         // Nach der Anwahl des Referenziertyps "Fliegendes Referenzieren", 
         // ein Zyklus später kann das Referenzieren gestartet
         IF (#siRefTypCyc = 0) THEN
           #siRefTypCyc := #siRefTypCyc + 1;
         ELSE
           // Referenzieren starten
           //#sxSendBuf.sxSTW1.RefStart := True;
           #sxSendBuf.STW1.%X11 := True;
         END_IF;
       END_IF;
     END_IF;
   ELSE
     // Werte wieder zurücknehmen
     (*#sxSendBuf.sxSTW1.Off1          := #Off1;
             #sxSendBuf.sxSTW1.RejTrvTsk     := False;
             #sxSendBuf.sxSTW1.TrvStart      := False;
             #sxSendBuf.sxEPosSTW1.MdiStart  := False;
             #sxSendBuf.sxSTW1.Jog1          := False;
             #sxSendBuf.sxSTW1.Jog2          := False;
             #sxSendBuf.sxEPosSTW1.MdiTyp    := False;
             #sxSendBuf.sxEPosSTW1.MdiPos    := False;
             #sxSendBuf.sxEPosSTW1.MdiNeg    := False;
             #sxSendBuf.sxEPosSTW1.MdiTrTyp  := False;
             #sxSendBuf.sxEPosSTW1.MdiSetup  := False;
             #sxSendBuf.sxEPosSTW2.SetRefPt  := False;
             #sxSendBuf.sxEPosSTW2.RefTyp    := False;
             #sxSendBuf.sxEPosSTW2.RefStDi   := False;
             #sxSendBuf.sxEPosSTW2.JogInc    := False;
             #sxSendBuf.sxSTW1.RefStart      := False;*)

     #sxSendBuf.STW1.%X0 := #EnableAxis;
     #sxSendBuf.STW1.%X4 := False;
     #sxSendBuf.STW1.%X6 := False;
     #sxSendBuf.EPosSTW1.%X15 := False;
     #sxSendBuf.STW1.%X8 := False;
     #sxSendBuf.STW1.%X9 := False;
     #sxSendBuf.EPosSTW1.%X8 := False;
     #sxSendBuf.EPosSTW1.%X9 := False;
     #sxSendBuf.EPosSTW1.%X10 := False;
     #sxSendBuf.EPosSTW1.%X12 := False;
     #sxSendBuf.EPosSTW1.%X14 := False;
     #sxSendBuf.EPosSTW2.%X1 := False;
     #sxSendBuf.EPosSTW2.%X8 := False;
     #sxSendBuf.EPosSTW2.%X9 := False;
     #sxSendBuf.EPosSTW2.%X5 := False;
     #sxSendBuf.STW1.%X11 := False;
   END_IF; // Hauptbetriebsart "Verfahrsätze" (Traversing Blocks)

   //Den Eingang ConfigEPos auf die einzelnen Bits im Telegramm verschalten
   #sxSendBuf.STW1.%X1 := #ConfigEPos.%X0;
   #sxSendBuf.STW1.%X2 := #ConfigEPos.%X1;
   #sxSendBuf.EPosSTW2.%X14 := #ConfigEPos.%X2;
   #sxSendBuf.EPosSTW2.%X15 := #ConfigEPos.%X3;
   #sxSendBuf.EPosSTW2.%X11 := #ConfigEPos.%X4;
   #sxSendBuf.EPosSTW2.%X10 := #ConfigEPos.%X5;
   #sxSendBuf.EPosSTW2.%X2 := #ConfigEPos.%X6;
   #sxSendBuf.STW1.%X13 := #ConfigEPos.%X7;
   #sxSendBuf.EPosSTW1.%X12 := #ConfigEPos.%X8;
   #sxSendBuf.STW2.%X0 := #ConfigEPos.%X9;
   #sxSendBuf.STW2.%X1 := #ConfigEPos.%X10;
   #sxSendBuf.STW2.%X2 := #ConfigEPos.%X11;
   #sxSendBuf.STW2.%X3 := #ConfigEPos.%X12;
   #sxSendBuf.STW2.%X4 := #ConfigEPos.%X13;
   #sxSendBuf.STW2.%X7 := #ConfigEPos.%X14;
   #sxSendBuf.STW1.%X12 := #ConfigEPos.%X15;
   #sxSendBuf.STW1.%X14 := #ConfigEPos.%X16;
   #sxSendBuf.STW1.%X15 := #ConfigEPos.%X17;
   #sxSendBuf.EPosSTW1.%X6 := #ConfigEPos.%X18;
   #sxSendBuf.EPosSTW1.%X7 := #ConfigEPos.%X19;
   #sxSendBuf.EPosSTW1.%X11 := #ConfigEPos.%X20;
   #sxSendBuf.EPosSTW1.%X13 := #ConfigEPos.%X21;
   #sxSendBuf.EPosSTW2.%X3 := #ConfigEPos.%X22;
   #sxSendBuf.EPosSTW2.%X4 := #ConfigEPos.%X23;
   #sxSendBuf.EPosSTW2.%X6 := #ConfigEPos.%X24;
   #sxSendBuf.EPosSTW2.%X7 := #ConfigEPos.%X25;
   #sxSendBuf.EPosSTW2.%X12 := #ConfigEPos.%X26;
   #sxSendBuf.EPosSTW2.%X13 := #ConfigEPos.%X27;
   #sxSendBuf.STW2.%X5 := #ConfigEPos.%X28;
   #sxSendBuf.STW2.%X6 := #ConfigEPos.%X29;
   #sxSendBuf.STW2.%X8 := #ConfigEPos.%X30;
   #sxSendBuf.STW2.%X9 := #ConfigEPos.%X31;


   #swSendBuf[0] := #sxSendBuf.STW1;
   #swSendBuf[1] := #sxSendBuf.EPosSTW1;
   #swSendBuf[2] := #sxSendBuf.EPosSTW2;
   #swSendBuf[3] := #sxSendBuf.STW2;
   #swSendBuf[4] := #sxSendBuf.OverrideV;
   #swSendBuf[5] := #sxSendBuf.Position.%W1;
   #swSendBuf[6] := #sxSendBuf.Position.%W0;
   #swSendBuf[7] := #sxSendBuf.Velocity.%W1;
   #swSendBuf[8] := #sxSendBuf.Velocity.%W0;
   #swSendBuf[9] := #sxSendBuf.OverrideA;
   #swSendBuf[10] := #sxSendBuf.OverrideD;
   #swSendBuf[11] := #sxSendBuf.Reserve;

   //Prozessdaten zur Signalbaugruppe schreiben
   #piRetSFC := DPWR_DAT(LADDR := #HWIDSTW,
                         RECORD := #swSendBuf);

   // Fehler der Rückmeldung ausgeben
   #DiagID := INT_TO_WORD(#piRetSFC);

   //kein Fehler beim Schreiben
   IF #piRetSFC = 0 THEN

     // Fehler wieder zurück nehmen
     IF (#swStatus = 16#8601) THEN
       #swStatus := 16#7002;
       #Error := False;
     END_IF;

     //Prozessdaten von der Signalbaugruppe lesen
     #piRetSFC := DPRD_DAT(LADDR := #HWIDZSW,
                           RECORD => #swRecvBuf);

     // Fehlermeldung der Rückmeldung ausgeben
     #DiagID := INT_TO_WORD(#piRetSFC);

     //Fehler beim Lesen (Profibus-Kommunikation unterbrochen)
     IF #piRetSFC <> 0 THEN

       // Fehler
       #Error := TRUE;
       #swStatus := 16#8600;

       // Zustandsworte löschen
       #sxRecvBuf.ZSW1 := W#16#0;
       #sxRecvBuf.EPosZSW1 := W#16#0;
       #sxRecvBuf.EPosZSW2 := W#16#0;
       #sxRecvBuf.ZSW2 := W#16#0;
       #sxRecvBuf.NotUsed := W#16#00;
       #sxRecvBuf.Position := DW#16#00;
       #sxRecvBuf.Velocity := DW#16#00;
       #sxRecvBuf.ErrNr := W#16#00;
       #sxRecvBuf.WarnNr := W#16#00;
       #sxRecvBuf.Reserve := W#16#00;

       // Werte auslesen
     ELSE

       // Fehler wieder zurück nehmen
       IF (#swStatus = 16#8600) THEN
         #swStatus := 16#7002;
         #Error := False;
       END_IF;

       #sxRecvBuf.ZSW1 := #swRecvBuf[0];
       #sxRecvBuf.EPosZSW1 := #swRecvBuf[1];
       #sxRecvBuf.EPosZSW2 := #swRecvBuf[2];
       #sxRecvBuf.ZSW2 := #swRecvBuf[3];
       #sxRecvBuf.NotUsed := #swRecvBuf[4];
       #sxRecvBuf.Position.%W1 := #swRecvBuf[5];
       #sxRecvBuf.Position.%W0 := #swRecvBuf[6];
       #sxRecvBuf.Velocity.%W1 := #swRecvBuf[7];
       #sxRecvBuf.Velocity.%W0 := #swRecvBuf[8];
       #sxRecvBuf.ErrNr := #swRecvBuf[9];
       #sxRecvBuf.WarnNr := #swRecvBuf[10];
       #sxRecvBuf.Reserve := #swRecvBuf[11];

       #aaa := INT_TO_REAL(WORD_TO_INT(#sxRecvBuf.Reserve));
       #bbb:=NORM_X_REAL(MAX := 16384.0, MIN := -16384.0, VALUE := #aaa);
       #Torque :=ABS(SCALE_X_REAL(MIN := #RefTorque*-1, MAX :=#RefTorque, VALUE := #bbb));

       // ZSW1 aufbereiten
       //#Busy := #sxRecvBuf.sxZSW1.IOp;
       #sbBusy := #sxRecvBuf.ZSW1.%X2;

       // Fehler auswerten
       IF #sxRecvBuf.ZSW1.%X3 THEN
           #swStatus := 16#8401;
         #Error := True;
       ELSIF #sxRecvBuf.ZSW1.%X6 THEN
         #swStatus := 16#8402;
         #Error := True;
       ELSE
         // Fehler wieder zurück nehmen
         IF (#swStatus = 16#8401) OR (#swStatus = 16#8402) THEN
           #swStatus := 16#7002;
           #Error := False;
         END_IF;
       END_IF;

       // EPOS_ZSW1            
       // EPOS-Wort-1 BIT 00 --> 1 = Active traversing block bit 0
       //IF #sxRecvBuf.sxEPosZSW1.ActTrvBit0 THEN
       IF #sxRecvBuf.EPosZSW1.%X0 THEN
         #swEPosZSW1 := #swEPosZSW1 OR W#16#01;
       ELSE
         #swEPosZSW1 := #swEPosZSW1 AND W#16#FFFE;
       END_IF;

       // EPOS-Wort-1 Bit 01 --> 1 = Active traversing block bit 1
       //IF #sxRecvBuf.sxEPosZSW1.ActTrvBit1 THEN
       IF #sxRecvBuf.EPosZSW1.%X1 THEN
         #swEPosZSW1 := #swEPosZSW1 OR W#16#02;
       ELSE
         #swEPosZSW1 := #swEPosZSW1 AND W#16#FFFD;
       END_IF;

       // EPOS-Wort-1 Bit 02 --> 1 = Active traversing block bit 2
       //IF #sxRecvBuf.sxEPosZSW1.ActTrvBit2 THEN
       IF #sxRecvBuf.EPosZSW1.%X2 THEN
         #swEPosZSW1 := #swEPosZSW1 OR W#16#04;
       ELSE
         #swEPosZSW1 := #swEPosZSW1 AND W#16#FFFB;
       END_IF;

       // EPOS-Wort-1 Bit 03 --> 1 = Active traversing block bit 3
       //IF #sxRecvBuf.sxEPosZSW1.ActTrvBit3 THEN
       IF #sxRecvBuf.EPosZSW1.%X3 THEN
         #swEPosZSW1 := #swEPosZSW1 OR W#16#08;
       ELSE
         #swEPosZSW1 := #swEPosZSW1 AND W#16#FFF7;
       END_IF;

       // EPOS-Wort-1 Bit 04 --> 1 = Active traversing block bit 4 
       //IF #sxRecvBuf.sxEPosZSW1.ActTrvBit4 THEN
       IF #sxRecvBuf.EPosZSW1.%X4 THEN
         #swEPosZSW1 := #swEPosZSW1 OR W#16#10;
       ELSE
         #swEPosZSW1 := #swEPosZSW1 AND W#16#FFEF;
       END_IF;

       // EPOS-Wort-1 Bit 05 --> 1 = Active traversing block bit 5
       //IF #sxRecvBuf.sxEPosZSW1.ActTrvBit5 THEN
       IF #sxRecvBuf.EPosZSW1.%X5 THEN
         #swEPosZSW1 := #swEPosZSW1 OR W#16#20;
       ELSE
         #swEPosZSW1 := #swEPosZSW1 AND W#16#FFDF;
       END_IF;

       // EPOS-Wort-1 Bit 08 --> 1 = STOP cam minus active
       //IF #sxRecvBuf.sxEPosZSW1.StpCamMinAct THEN
       IF #sxRecvBuf.EPosZSW1.%X8 THEN
         #swEPosZSW1 := #swEPosZSW1 OR W#16#100;
       ELSE
         #swEPosZSW1 := #swEPosZSW1 AND W#16#FEFF;
       END_IF;

       // EPOS-Wort-1 Bit 09 --> 1 = STOP cam plus active
       //IF #sxRecvBuf.sxEPosZSW1.StpCamPlsAct THEN
       IF #sxRecvBuf.EPosZSW1.%X9 THEN
         #swEPosZSW1 := #swEPosZSW1 OR W#16#200;
       ELSE
         #swEPosZSW1 := #swEPosZSW1 AND W#16#FDFF;
       END_IF;

       // EPOS-Wort-1 Bit 10 --> 1 = Jogging active
       //IF #sxRecvBuf.sxEPosZSW1.JogAct THEN
       IF #sxRecvBuf.EPosZSW1.%X10 THEN
         #swEPosZSW1 := #swEPosZSW1 OR W#16#400;
       ELSE
         #swEPosZSW1 := #swEPosZSW1 AND W#16#FBFF;
       END_IF;

       // EPOS-Wort-1 Bit 11 --> 1 = Reference point approach active
       //IF #sxRecvBuf.sxEPosZSW1.RefAct THEN
       IF #sxRecvBuf.EPosZSW1.%X11 THEN
         #swEPosZSW1 := #swEPosZSW1 OR W#16#800;
       ELSE
         #swEPosZSW1 := #swEPosZSW1 AND W#16#F7FF;
       END_IF;

       // Anstossen des fliegenden Referenzieren prüfen, wenn die Rückmeldung fehlt dann wiederholen
       //IF NOT #sxRecvBuf.sxEPosZSW1.FlyRefAct AND #sbRefTyp AND #sxSendBuf.sxSTW1.RefStart THEN
       IF NOT #sxRecvBuf.EPosZSW1.%X12 AND #sbRefTyp AND #sxSendBuf.STW1.%X11 THEN

         // Wiederholung anstossen 
         IF #siRefActRetry < #siRetryMax THEN
           #siRefActRetry := #siRefActRetry + 1;

           // Referenzieren starten wieder wegnehmen
           //#sxSendBuf.sxSTW1.RefStart := False;
           #sxSendBuf.STW1.%X11 := False;
         ELSE

           // Fehlermeldung
           #swStatus := 16#8403;
           #Error := True;
         END_IF;
       ELSE

         // Fehler wieder zurücknehmen, wenn er mal ausgelöst wurde
         IF #swStatus = 16#8403 THEN
           #swStatus := 16#7002;
           #Error := False;
         END_IF;
         // Zähler zurücksetzen bei Rückmeldung fliegendes Referenzieren jetzt aktiviert oder bei Abwahl der Funktion
         IF (#sxRecvBuf.EPosZSW1.%X12 AND #sbRefTyp AND #sxSendBuf.STW1.%X11) OR NOT #FlyRef THEN
           #siRefActRetry := 0;
         END_IF;
       END_IF;

       // EPOS-Wort-1 Bit 12 --> 1 = Flying referencing active
       //IF #sxRecvBuf.sxEPosZSW1.FlyRefAct THEN
       IF #sxRecvBuf.EPosZSW1.%X12 THEN
         #swEPosZSW1 := #swEPosZSW1 OR W#16#1000;
       ELSE
         #swEPosZSW1 := #swEPosZSW1 AND W#16#EFFF;
       END_IF;

       // EPOS-Wort-1 Bit 13 --> 1 = Traversing block active
       //IF #sxRecvBuf.sxEPosZSW1.TrvBlAct THEN
       IF #sxRecvBuf.EPosZSW1.%X13 THEN
         #swEPosZSW1 := #swEPosZSW1 OR W#16#2000;
       ELSE
         #swEPosZSW1 := #swEPosZSW1 AND W#16#DFFF;
       END_IF;

       // EPOS-Wort-1 Bit 14 --> 1 = MDI setup active
       //IF #sxRecvBuf.sxEPosZSW1.MdiStupAct THEN
       IF #sxRecvBuf.EPosZSW1.%X14 THEN
         #swEPosZSW1 := #swEPosZSW1 OR W#16#4000;
       ELSE
         #swEPosZSW1 := #swEPosZSW1 AND W#16#BFFF;
       END_IF;

       // EPOS-Wort-1 Bit 15 --> 1 = MDI positing active
       //IF #sxRecvBuf.sxEPosZSW1.MdiPosAct THEN
       IF #sxRecvBuf.EPosZSW1.%X15 THEN
         #swEPosZSW1 := #swEPosZSW1 OR W#16#8000;
       ELSE
         #swEPosZSW1 := #swEPosZSW1 AND W#16#7FFF;
       END_IF;

       // EPOS_ZSW2 
       // EPOS-Wort-2 Bit 00 --> 1 = Tracking mode active
       //IF #sxRecvBuf.sxEPosZSW2.TrkModeAct THEN
       IF #sxRecvBuf.EPosZSW2.%X0 THEN
         #swEPosZSW2 := #swEPosZSW2 OR W#16#01;
       ELSE
         #swEPosZSW2 := #swEPosZSW2 AND W#16#FFFE;
       END_IF;

       // EPOS-Wort-2 Bit 01 --> 1 = Velocity limit active
       //IF #sxRecvBuf.sxEPosZSW2.VeloLimAct THEN
       IF #sxRecvBuf.EPosZSW2.%X1 THEN
         #swEPosZSW2 := #swEPosZSW2 OR W#16#02;
       ELSE
         #swEPosZSW2 := #swEPosZSW2 AND W#16#FFFD;
       END_IF;

       // EPOS-Wort-2 Bit 02 --> 1 = Setpoint static
       //IF #sxRecvBuf.sxEPosZSW2.SetPStat THEN
       IF #sxRecvBuf.EPosZSW2.%X2 THEN
         #swEPosZSW2 := #swEPosZSW2 OR W#16#04;
       ELSE
         #swEPosZSW2 := #swEPosZSW2 AND W#16#FFFB;
       END_IF;

       // EPOS-Wort-2 Bit 03 --> 1 = Printmark outside outer window
       //IF #sxRecvBuf.sxEPosZSW2.PrnMrkOut THEN
       IF #sxRecvBuf.EPosZSW2.%X3 THEN
         #swEPosZSW2 := #swEPosZSW2 OR W#16#08;
       ELSE
         #swEPosZSW2 := #swEPosZSW2 AND W#16#FFF7;
       END_IF;

       // EPOS-Wort-2 Bit 04 --> 1 = Axis forwards
       //IF #sxRecvBuf.sxEPosZSW2.FWD THEN
       IF #sxRecvBuf.EPosZSW2.%X4 THEN
         #swEPosZSW2 := #swEPosZSW2 OR W#16#10;
       ELSE
         #swEPosZSW2 := #swEPosZSW2 AND W#16#FFEF;
       END_IF;

       // EPOS-Wort-2 Bit 05 --> 1 = Axis backwards
       //IF #sxRecvBuf.sxEPosZSW2.BWD THEN
       IF #sxRecvBuf.EPosZSW2.%X5 THEN
         #swEPosZSW2 := #swEPosZSW2 OR W#16#20;
       ELSE
         #swEPosZSW2 := #swEPosZSW2 AND W#16#FFDF;
       END_IF;

       // EPOS-Wort-2 Bit 06 --> 1 = Software limit switch minus active
       //IF #sxRecvBuf.sxEPosZSW2.SftSwMinAct THEN
       IF #sxRecvBuf.EPosZSW2.%X6 THEN
         #swEPosZSW2 := #swEPosZSW2 OR W#16#40;
       ELSE
         #swEPosZSW2 := #swEPosZSW2 AND W#16#FFBF;
       END_IF;

       // EPOS-Wort-2 Bit 07 --> 1 = Software limit switch plus active
       //IF #sxRecvBuf.sxEPosZSW2.SftSwPlsAct THEN
       IF #sxRecvBuf.EPosZSW2.%X7 THEN
         #swEPosZSW2 := #swEPosZSW2 OR W#16#80;
       ELSE
         #swEPosZSW2 := #swEPosZSW2 AND W#16#FF7F;
       END_IF;

       // EPOS-Wort-2 Bit 08 --> 1 = Position actual value <= cam position 1
       //IF #sxRecvBuf.sxEPosZSW2.PosSmCam1 THEN
       IF #sxRecvBuf.EPosZSW2.%X8 THEN
         #swEPosZSW2 := #swEPosZSW2 OR W#16#100;
       ELSE
         #swEPosZSW2 := #swEPosZSW2 AND W#16#FEFF;
       END_IF;

       // EPOS-Wort-2 Bit 09 --> 1 = Position actual value <= cam position 2
       //IF #sxRecvBuf.sxEPosZSW2.PosSmCam2 THEN
       IF #sxRecvBuf.EPosZSW2.%X9 THEN
         #swEPosZSW2 := #swEPosZSW2 OR W#16#200;
       ELSE
         #swEPosZSW2 := #swEPosZSW2 AND W#16#FDFF;
       END_IF;

       // EPOS-Wort-2 Bit 10 --> 1 = Direct output 1 via traversing block
       //IF #sxRecvBuf.sxEPosZSW2.TrvOut1 THEN
       IF #sxRecvBuf.EPosZSW2.%X10 THEN
         #swEPosZSW2 := #swEPosZSW2 OR W#16#400;
       ELSE
         #swEPosZSW2 := #swEPosZSW2 AND W#16#FBFF;
       END_IF;

       // EPOS-Wort-2 Bit 11 --> 1 = Direct output 2 via traversing block
       //IF #sxRecvBuf.sxEPosZSW2.TrvOut2 THEN
       IF #sxRecvBuf.EPosZSW2.%X11 THEN
         #swEPosZSW2 := #swEPosZSW2 OR W#16#800;
       ELSE
         #swEPosZSW2 := #swEPosZSW2 AND W#16#F7FF;
       END_IF;

       // EPOS-Wort-2 Bit 12 --> 1 = Fixed STOP reached
       //IF #sxRecvBuf.sxEPosZSW2.FxStpRd THEN
       IF #sxRecvBuf.EPosZSW2.%X12 THEN
         #swEPosZSW2 := #swEPosZSW2 OR W#16#1000;
       ELSE
         #swEPosZSW2 := #swEPosZSW2 AND W#16#EFFF;
       END_IF;

       // EPOS-Wort-2 Bit 13 --> 1 = Fixed STOP clamping torque reached
       //IF #sxRecvBuf.sxEPosZSW2.FxStpTrRd THEN
       IF #sxRecvBuf.EPosZSW2.%X13 THEN
         #swEPosZSW2 := #swEPosZSW2 OR W#16#2000;
       ELSE
         #swEPosZSW2 := #swEPosZSW2 AND W#16#DFFF;
       END_IF;

       // EPOS-Wort-2 Bit 14 --> 1 = Traversing fixed STOP active
       //IF #sxRecvBuf.sxEPosZSW2.TrvFxStpAct THEN
       IF #sxRecvBuf.EPosZSW2.%X14 THEN
         #swEPosZSW2 := #swEPosZSW2 OR W#16#4000;
       ELSE
         #swEPosZSW2 := #swEPosZSW2 AND W#16#BFFF;
       END_IF;

       // EPOS-Wort-2 Bit 15 --> 1 = Traversing command active
       //IF #sxRecvBuf.sxEPosZSW2.CmdAct THEN
       IF #sxRecvBuf.EPosZSW2.%X15 THEN
         #swEPosZSW2 := #swEPosZSW2 OR W#16#8000;
       ELSE
         #swEPosZSW2 := #swEPosZSW2 AND W#16#7FFF;
       END_IF;

       #sbReady := #sxRecvBuf.ZSW1.%X1;

       #AxisEnabled := #sxRecvBuf.ZSW1.%X2;
       #sbIOp := #sxRecvBuf.ZSW1.%X2;

       #AxisError := #sxRecvBuf.ZSW1.%X3;
       #sbFault := #sxRecvBuf.ZSW1.%X3;

       #AxisWarn := #sxRecvBuf.ZSW1.%X7;
       #sbAlarm := #sxRecvBuf.ZSW1.%X7;

       #AxisPosOk := #sxRecvBuf.ZSW1.%X10;
       #AxisRef := #sxRecvBuf.ZSW1.%X11;
       #AxisSpFixed := #sxRecvBuf.ZSW1.%X13;

       #sbAccel := #sxRecvBuf.ZSW1.%X14;
       #sbDecel := #sxRecvBuf.ZSW1.%X15;

       //#ActVelocity := DWORD_TO_DINT(#sxRecvBuf.Velocity);
       #v1 := DINT_TO_REAL(DWORD_TO_DINT(#sxRecvBuf.Velocity));
       #v2:=(#v1+16#40000000) / 16#80000000;
       #ActVelocity := ABS(SCALE_X_REAL(MIN := -1*#RefSpeed, MAX := #RefSpeed, VALUE := #v2));

       //#ActPosition := DWORD_TO_DINT(#sxRecvBuf.Position);
       #ActPosition :=(DINT_TO_REAL(DWORD_TO_DINT(#sxRecvBuf.Position)) / #Factor);


       #ActMode := #ModePos;
       #ActWarn := #sxRecvBuf.WarnNr;
       #ActFault := #sxRecvBuf.ErrNr;

       #Lockout := #sxRecvBuf.ZSW1.%X6;
       //Soft Positio OK
       IF ABS_REAL(#Position - #ActPosition) < #SoftPosTlr THEN
           ;
           #SoftPosOK := TRUE;
       ELSE
           #SoftPosOK := FALSE;
       END_IF;
     END_IF;
   ELSE

     // Fehler
     #Error := TRUE;
     #swStatus := 16#8601;

   END_IF;

   // Initialisierung von Ausg㭧en
   #Status := #swStatus;
   #EPosZSW1 := #swEPosZSW1;
   #EPosZSW2 := #swEPosZSW2;
END_FUNCTION_BLOCK

// ===== library: MasterCopy "ServoAxisV90" =====

// folder: AxisControl

FUNCTION_BLOCK "ServoAxisV90"   // FB602, LAD
{ S7_Optimized_Access := 'TRUE' }
VERSION : 0.1
   VAR_INPUT
      HwID : HW_IO;
      "Enb?" : Bool;
      iLLim : Bool;
      iHLim : Bool;
      iMotionPermit : Bool;
      iJogPermit : Bool;
      iReset : Bool;
      bwPos : Real := 0.0;   // Geri Pozisyon Bilgisi
      fwPos : Real := 0.0;   // İleri Pozisyon Bilgisi
      bwTol : Real := 0.0;   // İleride Bilgisi Toleransı
      fwTol : Real := 0.0;   // Geride Bilgisi Toleransı
      inSpeed : Real;
   END_VAR
   VAR_OUTPUT
      qBrake : Bool;
   END_VAR
   VAR_IN_OUT
      ManCmd : "ManServo";
      iHoldingOff : Bool;
   END_VAR
   VAR
      Servo : "SINA_POS";
      AutoCmd : Struct
         Go1TargetPos : Bool;
         Go2TargetPos : Bool;
         Go3TargetPos : Bool;
         Go1WaitingPos : Bool;
         Go2WaitingPos : Bool;
         Go3WaitingPos : Bool;
         Go4WaitingPos : Bool;
         TargetPos : Real;
         WaitingPos : Real;
         Speed : Int;
      END_STRUCT;
      Auto : Struct
         GoAbs : Bool;
         "Step" : Int;
      END_STRUCT;
      Man : Struct
         GoAbs : Bool;
         "Step" : Int;
      END_STRUCT;
      Homing : Struct
         Execute : Bool;
         "Step" : Int;
      END_STRUCT;
      Ready : Bool;
      OnSafetyArea : Bool;
      PosOK : Bool;
      OnBwPos : Bool;
      OnFwPos : Bool;
      OnBw2Pos : Bool;
      mAxisMoving : Bool;
      PosTemp : Real;
      "Timer" : Struct
         T1 : IEC_TIMER;
         T2 : IEC_TIMER;
         T3 : IEC_TIMER;
         T4 : IEC_TIMER;
         T5 : IEC_TIMER;
         T6 : IEC_TIMER;
         T7 : IEC_TIMER;
         T8 : IEC_TIMER;
         T9 : IEC_TIMER;
         T10 : IEC_TIMER;
         T11 : IEC_TIMER;
      END_STRUCT;
      Alarm : Struct
         PermissionErr : Bool;
         EnbErr : Bool;
      END_STRUCT;
      negBwTol : Real;
      p_trg : Array[0..3] of Bool;
      negFwTol : Real;
      ovDec : Int;
   END_VAR
   VAR_TEMP
      Temp1 : Real;
      Temp2 : Real;
      temp3 : Real;
   END_VAR
   VAR_TEMP   // added for the SCL form of the ladder/FBD networks
      _w1 : Bool;
      _w2 : Bool;
      _w3 : Bool;
      _w4 : Bool;
   END_VAR
BEGIN

REGION Network 1: Sina Pos Block
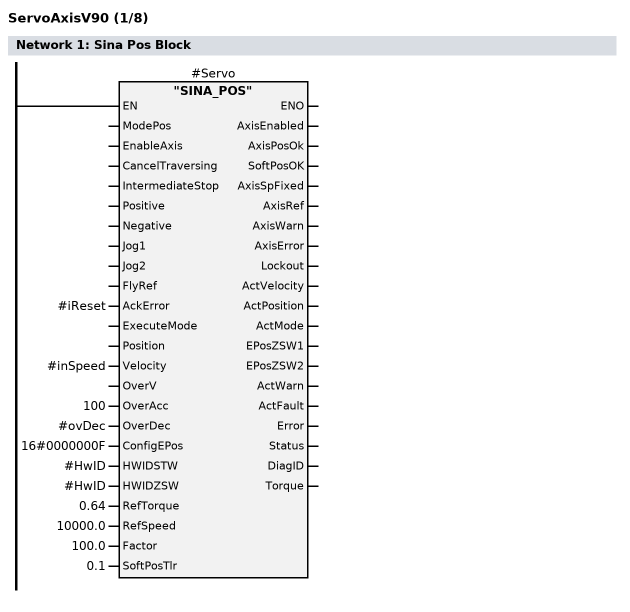
   RUNG wire#powerrail
      #Servo(ModePos :=, EnableAxis :=, CancelTraversing :=, IntermediateStop :=, Positive :=, Negative :=, Jog1 :=, Jog2 :=, FlyRef :=, AckError := #iReset, ExecuteMode :=, Position :=, Velocity := #inSpeed, OverV :=, OverAcc := 100, OverDec := #ovDec, ConfigEPos := 16#0000000F, HWIDSTW := #HwID, HWIDZSW := #HwID, RefTorque := 0.64, RefSpeed := 10000.0, Factor := 100.0, SoftPosTlr := 0.1, AxisEnabled =>, AxisPosOk =>, SoftPosOK =>, AxisSpFixed =>, AxisRef =>, AxisWarn =>, AxisError =>, Lockout =>, ActVelocity =>, ActPosition =>, ActMode =>, EPosZSW1 =>, EPosZSW2 =>, ActWarn =>, ActFault =>, Error =>, Status =>, DiagID =>, Torque =>)
   END_RUNG
   // the same network as SCL:
   #Servo(AckError := #iReset,   // "SINA_POS"
          Velocity := #inSpeed,
          OverAcc := 100,
          OverDec := #ovDec,
          ConfigEPos := 16#0000000F,
          HWIDSTW := #HwID,
          HWIDZSW := #HwID,
          RefTorque := 0.64,
          RefSpeed := 10000.0,
          Factor := 100.0,
          SoftPosTlr := 0.1);
END_REGION

REGION Network 2: Drive On
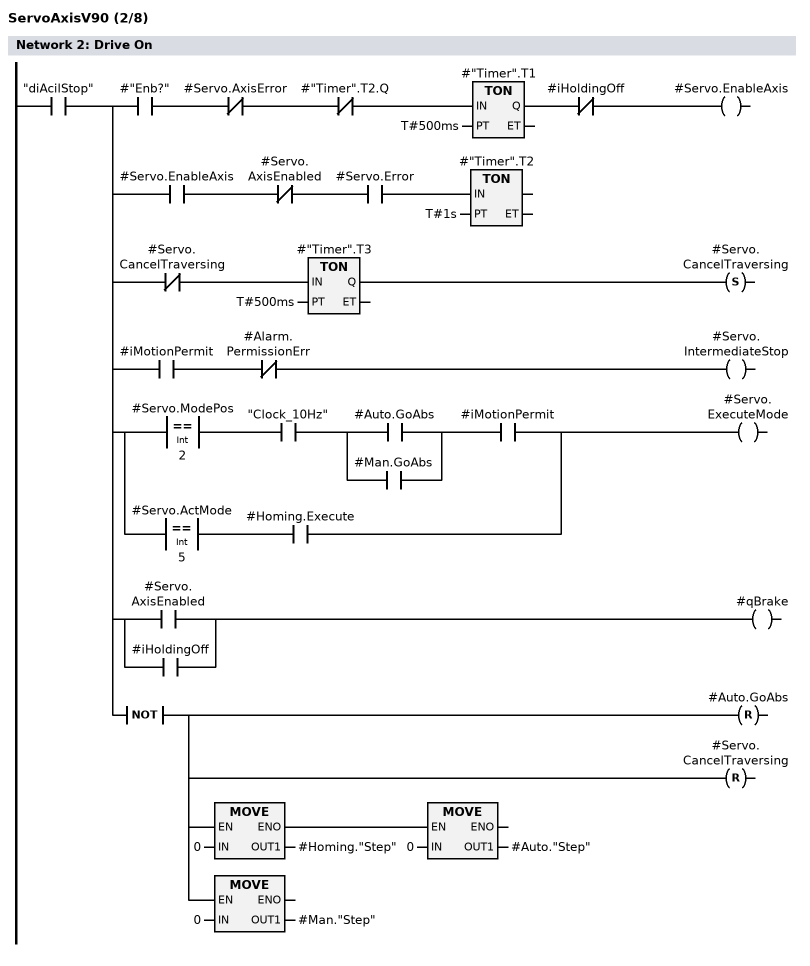
   // ENO of a box is taken as its EN; it also drops when the box reports an error
   #"Timer".T1.TON(IN := "diAcilStop" AND #"Enb?" AND NOT #Servo.AxisError AND NOT #"Timer".T2.Q, PT := T#500ms);
   #Servo.EnableAxis := #"Timer".T1.Q AND NOT #iHoldingOff;
   #"Timer".T2.TON(IN := "diAcilStop" AND #Servo.EnableAxis AND NOT #Servo.AxisEnabled AND #Servo.Error,
                   PT := T#1s);
   #"Timer".T3.TON(IN := "diAcilStop" AND NOT #Servo.CancelTraversing, PT := T#500ms);
   IF #"Timer".T3.Q THEN #Servo.CancelTraversing := TRUE; END_IF;
   #Servo.IntermediateStop := "diAcilStop" AND #iMotionPermit AND NOT #Alarm.PermissionErr;
   #Servo.ExecuteMode := "diAcilStop" AND (((#Servo.ModePos = 2) AND "Clock_10Hz" AND (#Auto.GoAbs OR #Man.GoAbs) AND #iMotionPermit) OR ((#Servo.ActMode = 5) AND #Homing.Execute));
   #qBrake := "diAcilStop" AND (#Servo.AxisEnabled OR #iHoldingOff);
   IF NOT "diAcilStop" THEN
       #Auto.GoAbs := FALSE;
       #Servo.CancelTraversing := FALSE;
       #Homing."Step" := 0;
       #Auto."Step" := 0;
       #Man."Step" := 0;
   END_IF;
END_REGION

REGION Network 3: On Safety Area & Servo Ready
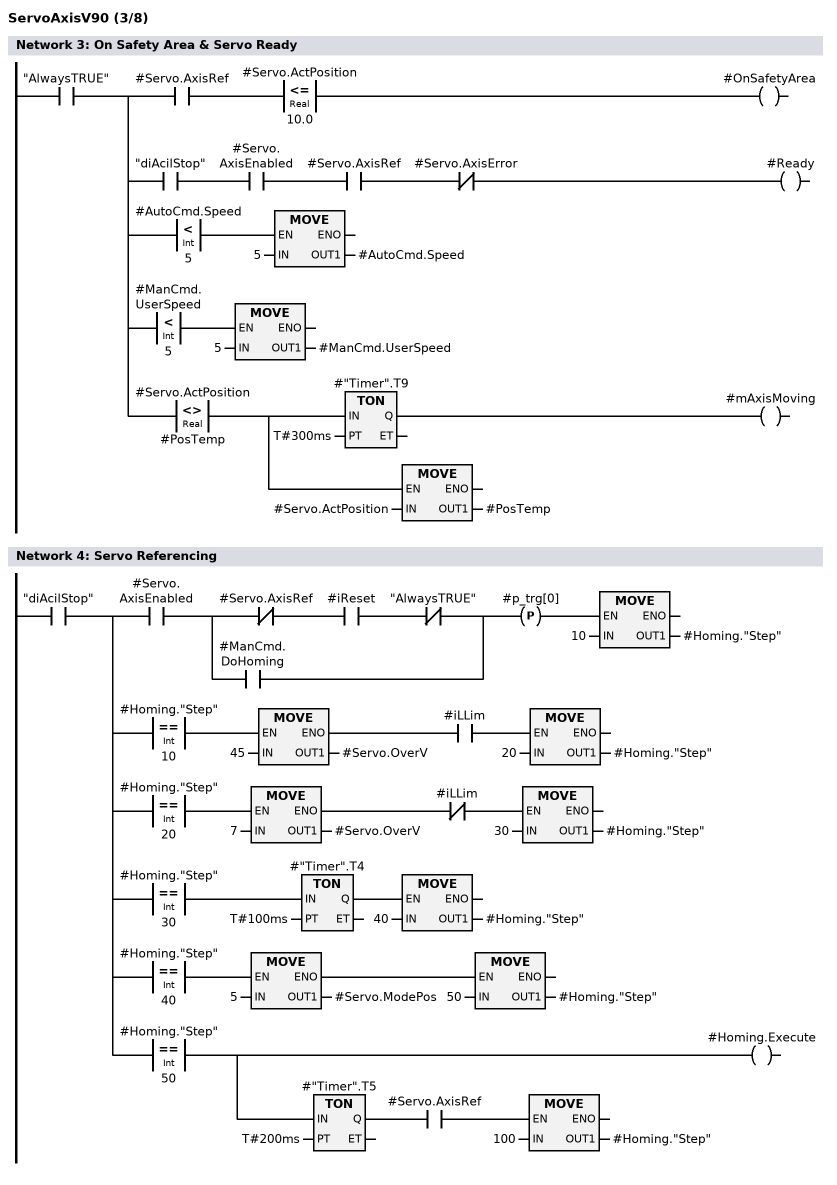
   #OnSafetyArea := "AlwaysTRUE" AND #Servo.AxisRef AND (#Servo.ActPosition <= 10.0);
   #Ready := "AlwaysTRUE" AND "diAcilStop" AND #Servo.AxisEnabled AND #Servo.AxisRef AND NOT #Servo.AxisError;
   IF "AlwaysTRUE" AND (#AutoCmd.Speed < 5) THEN #AutoCmd.Speed := 5; END_IF;
   IF "AlwaysTRUE" AND (#ManCmd.UserSpeed < 5) THEN #ManCmd.UserSpeed := 5; END_IF;
   #_w1 := "AlwaysTRUE" AND (#Servo.ActPosition <> #PosTemp);
   #"Timer".T9.TON(IN := #_w1, PT := T#300ms);
   #mAxisMoving := #"Timer".T9.Q;
   IF #_w1 THEN #PosTemp := #Servo.ActPosition; END_IF;
END_REGION

REGION Network 4: Servo Referencing
   // ENO of a box is taken as its EN; it also drops when the box reports an error
   #_w1 := "diAcilStop" AND #Servo.AxisEnabled AND ((NOT #Servo.AxisRef AND #iReset AND NOT "AlwaysTRUE") OR #ManCmd.DoHoming);
   #_w2 := #_w1 AND NOT #p_trg[0];   // rising edge
   #p_trg[0] := #_w1;
   IF #_w2 THEN #Homing."Step" := 10; END_IF;
   #_w3 := "diAcilStop" AND (#Homing."Step" = 10);
   IF #_w3 THEN #Servo.OverV := 45; END_IF;
   IF #_w3 AND #iLLim THEN #Homing."Step" := 20; END_IF;
   #_w4 := "diAcilStop" AND (#Homing."Step" = 20);
   IF #_w4 THEN #Servo.OverV := 7; END_IF;
   IF #_w4 AND NOT #iLLim THEN #Homing."Step" := 30; END_IF;
   #"Timer".T4.TON(IN := "diAcilStop" AND (#Homing."Step" = 30), PT := T#100ms);
   IF #"Timer".T4.Q THEN #Homing."Step" := 40; END_IF;
   IF "diAcilStop" AND (#Homing."Step" = 40) THEN
       #Servo.ModePos := 5;
       #Homing."Step" := 50;
   END_IF;
   #Homing.Execute := "diAcilStop" AND (#Homing."Step" = 50);
   #"Timer".T5.TON(IN := #Homing.Execute, PT := T#200ms);
   IF #"Timer".T5.Q AND #Servo.AxisRef THEN #Homing."Step" := 100; END_IF;
END_REGION

REGION Network 5: Jogging
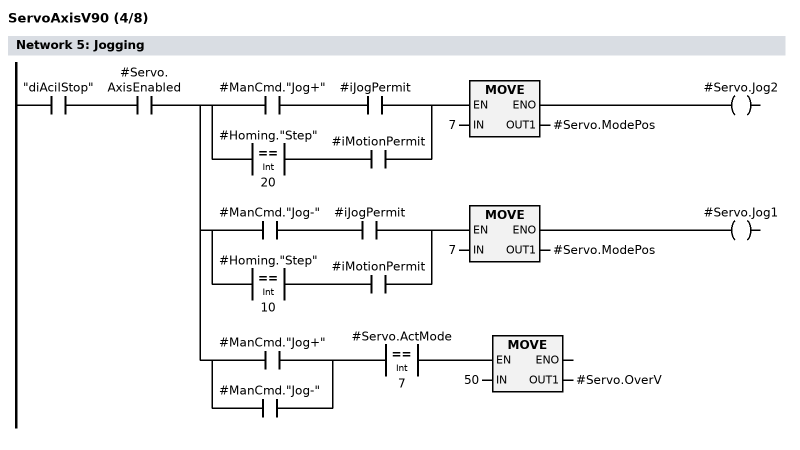
   RUNG wire#powerrail
      Contact( "diAcilStop" )
      Contact( #Servo.AxisEnabled )
      wire#w1
      Contact( #ManCmd."Jog+" )
      Contact( #iJogPermit )
      wire#w2
      { S7_GenerateENO := "TRUE" } Move(in := 7, out1 => #Servo.ModePos)
      Coil( #Servo.Jog2 )
   END_RUNG
   RUNG wire#w1
      { S7_Templates := "SrcType := Int" } EQ_Contact(in1 := #Homing."Step", in2 := 20)
      Contact( #iMotionPermit )
   END_RUNG wire#w2
   RUNG wire#w1
      Contact( #ManCmd."Jog-" )
      Contact( #iJogPermit )
      wire#w3
      { S7_GenerateENO := "TRUE" } Move(in := 7, out1 => #Servo.ModePos)
      Coil( #Servo.Jog1 )
   END_RUNG
   RUNG wire#w1
      { S7_Templates := "SrcType := Int" } EQ_Contact(in1 := #Homing."Step", in2 := 10)
      Contact( #iMotionPermit )
   END_RUNG wire#w3
   RUNG wire#w1
      Contact( #ManCmd."Jog+" )
      wire#w4
      { S7_Templates := "SrcType := Int" } EQ_Contact(in1 := #Servo.ActMode, in2 := 7)
      { S7_GenerateENO := "TRUE" } Move(in := 50, out1 => #Servo.OverV)
   END_RUNG
   RUNG wire#w1
      Contact( #ManCmd."Jog-" )
   END_RUNG wire#w4
   // the same network as SCL:
   // ENO of a box is taken as its EN; it also drops when the box reports an error
   #_w1 := "diAcilStop" AND #Servo.AxisEnabled;
   #_w2 := #_w1 AND ((#ManCmd."Jog+" AND #iJogPermit) OR ((#Homing."Step" = 20) AND #iMotionPermit));
   IF #_w2 THEN #Servo.ModePos := 7; END_IF;
   #Servo.Jog2 := #_w2;
   #_w3 := #_w1 AND ((#ManCmd."Jog-" AND #iJogPermit) OR ((#Homing."Step" = 10) AND #iMotionPermit));
   IF #_w3 THEN #Servo.ModePos := 7; END_IF;
   #Servo.Jog1 := #_w3;
   IF #_w1 AND (#ManCmd."Jog+" OR #ManCmd."Jog-") AND (#Servo.ActMode = 7) THEN #Servo.OverV := 50; END_IF;
END_REGION

REGION Network 6: Automatic Motion
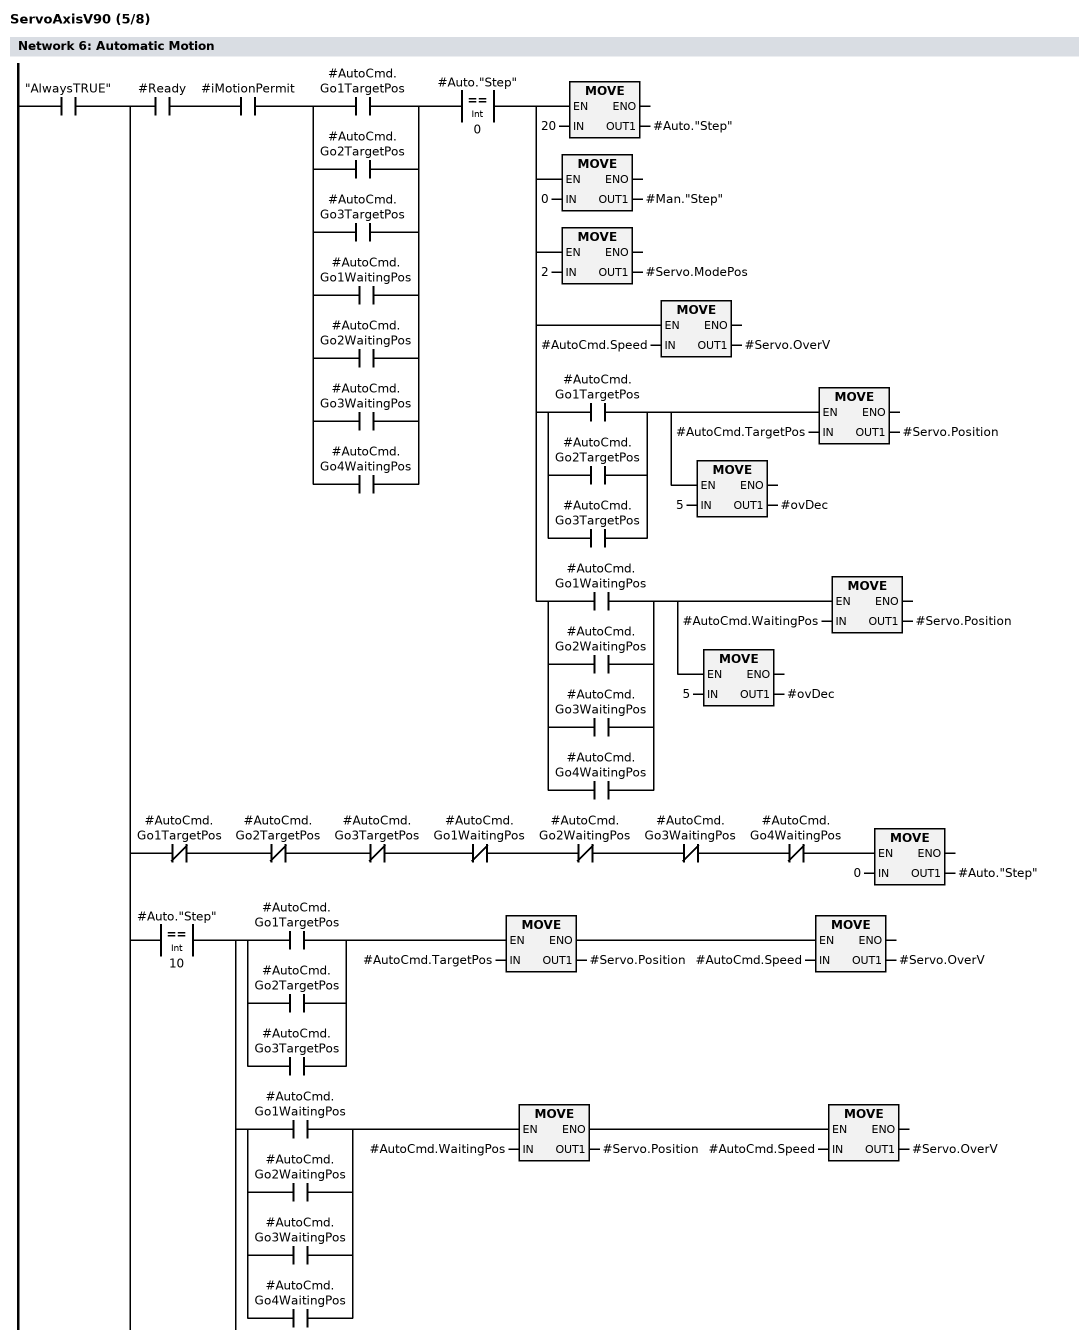
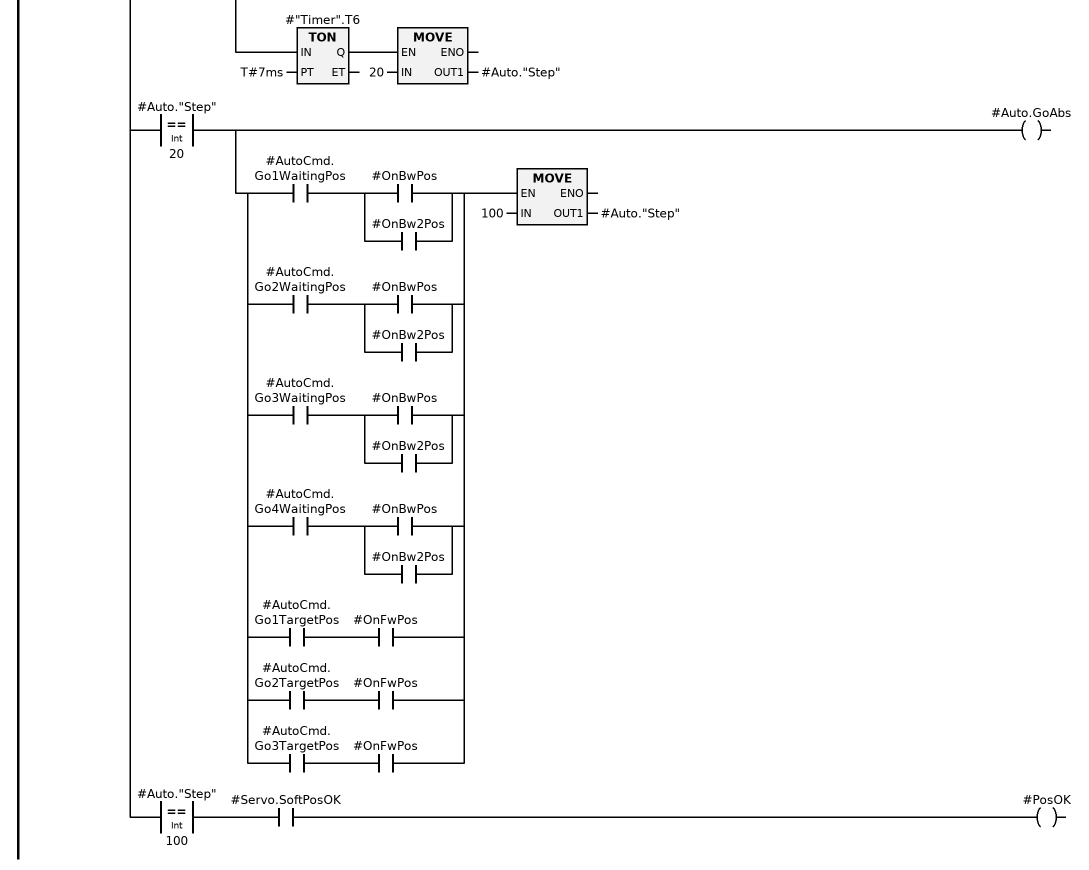
   // ENO of a box is taken as its EN; it also drops when the box reports an error
   #_w1 := "AlwaysTRUE" AND #Ready AND #iMotionPermit AND (#AutoCmd.Go1TargetPos OR #AutoCmd.Go2TargetPos OR #AutoCmd.Go3TargetPos OR #AutoCmd.Go1WaitingPos OR #AutoCmd.Go2WaitingPos OR #AutoCmd.Go3WaitingPos OR #AutoCmd.Go4WaitingPos) AND (#Auto."Step" = 0);
   IF #_w1 THEN
       #Auto."Step" := 20;
       #Man."Step" := 0;
       #Servo.ModePos := 2;
       #Servo.OverV := #AutoCmd.Speed;
   END_IF;
   IF #_w1 AND (#AutoCmd.Go1TargetPos OR #AutoCmd.Go2TargetPos OR #AutoCmd.Go3TargetPos) THEN
       #Servo.Position := #AutoCmd.TargetPos;
       #ovDec := 5;
   END_IF;
   IF #_w1 AND (#AutoCmd.Go1WaitingPos OR #AutoCmd.Go2WaitingPos OR #AutoCmd.Go3WaitingPos OR #AutoCmd.Go4WaitingPos) THEN
       #Servo.Position := #AutoCmd.WaitingPos;
       #ovDec := 5;
   END_IF;
   IF "AlwaysTRUE" AND NOT #AutoCmd.Go1TargetPos AND NOT #AutoCmd.Go2TargetPos AND NOT #AutoCmd.Go3TargetPos AND NOT #AutoCmd.Go1WaitingPos AND NOT #AutoCmd.Go2WaitingPos AND NOT #AutoCmd.Go3WaitingPos AND NOT #AutoCmd.Go4WaitingPos THEN
       #Auto."Step" := 0;
   END_IF;
   #_w2 := "AlwaysTRUE" AND (#Auto."Step" = 10);
   IF #_w2 AND (#AutoCmd.Go1TargetPos OR #AutoCmd.Go2TargetPos OR #AutoCmd.Go3TargetPos) THEN
       #Servo.Position := #AutoCmd.TargetPos;
       #Servo.OverV := #AutoCmd.Speed;
   END_IF;
   IF #_w2 AND (#AutoCmd.Go1WaitingPos OR #AutoCmd.Go2WaitingPos OR #AutoCmd.Go3WaitingPos OR #AutoCmd.Go4WaitingPos) THEN
       #Servo.Position := #AutoCmd.WaitingPos;
       #Servo.OverV := #AutoCmd.Speed;
   END_IF;
   #"Timer".T6.TON(IN := #_w2, PT := T#7ms);
   IF #"Timer".T6.Q THEN #Auto."Step" := 20; END_IF;
   #Auto.GoAbs := "AlwaysTRUE" AND (#Auto."Step" = 20);
   IF #Auto.GoAbs AND ((#AutoCmd.Go1WaitingPos AND (#OnBwPos OR #OnBw2Pos)) OR (#AutoCmd.Go2WaitingPos AND (#OnBwPos OR #OnBw2Pos)) OR (#AutoCmd.Go3WaitingPos AND (#OnBwPos OR #OnBw2Pos)) OR (#AutoCmd.Go4WaitingPos AND (#OnBwPos OR #OnBw2Pos)) OR (#AutoCmd.Go1TargetPos AND #OnFwPos) OR (#AutoCmd.Go2TargetPos AND #OnFwPos) OR (#AutoCmd.Go3TargetPos AND #OnFwPos)) THEN
       #Auto."Step" := 100;
   END_IF;
   #PosOK := "AlwaysTRUE" AND (#Auto."Step" = 100) AND #Servo.SoftPosOK;
END_REGION

REGION Network 7: Manuel Motion
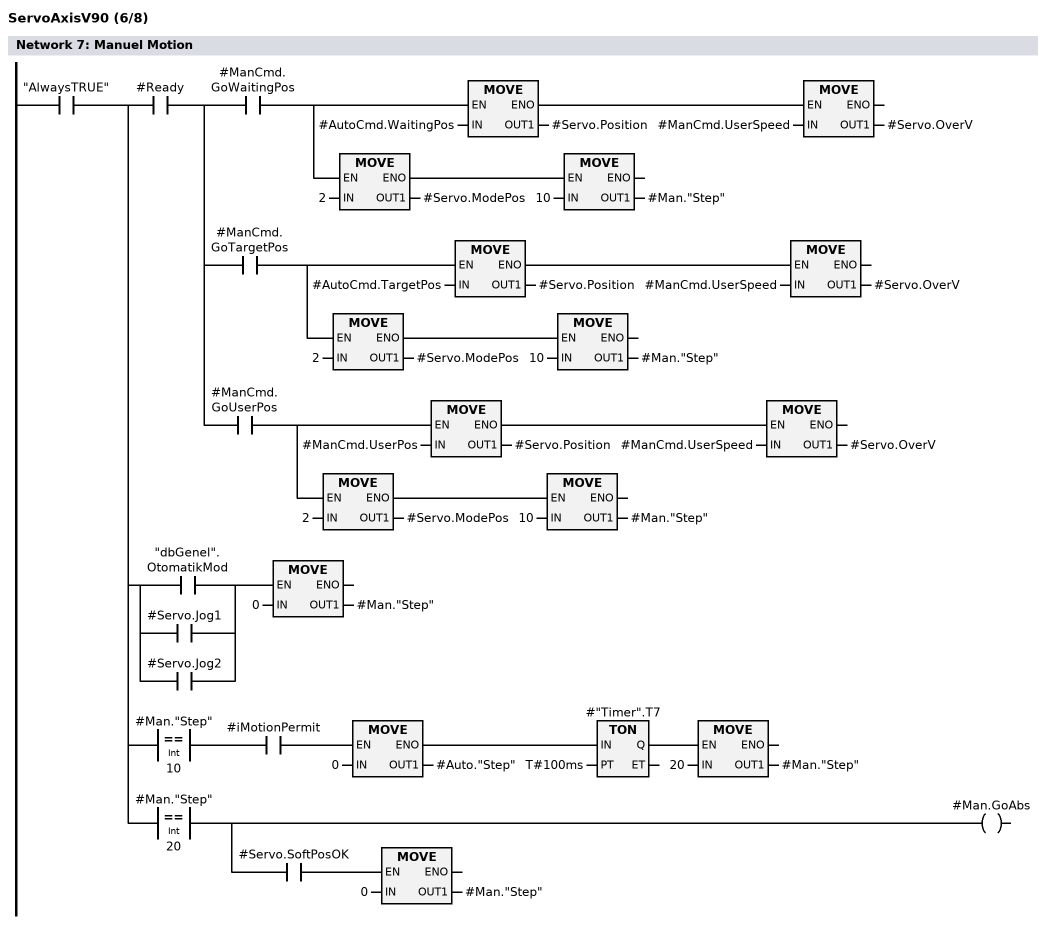
   // ENO of a box is taken as its EN; it also drops when the box reports an error
   #_w1 := "AlwaysTRUE" AND #Ready;
   IF #_w1 AND #ManCmd.GoWaitingPos THEN
       #Servo.Position := #AutoCmd.WaitingPos;
       #Servo.OverV := #ManCmd.UserSpeed;
       #Servo.ModePos := 2;
       #Man."Step" := 10;
   END_IF;
   IF #_w1 AND #ManCmd.GoTargetPos THEN
       #Servo.Position := #AutoCmd.TargetPos;
       #Servo.OverV := #ManCmd.UserSpeed;
       #Servo.ModePos := 2;
       #Man."Step" := 10;
   END_IF;
   IF #_w1 AND #ManCmd.GoUserPos THEN
       #Servo.Position := #ManCmd.UserPos;
       #Servo.OverV := #ManCmd.UserSpeed;
       #Servo.ModePos := 2;
       #Man."Step" := 10;
   END_IF;
   IF "AlwaysTRUE" AND ("dbGenel".OtomatikMod OR #Servo.Jog1 OR #Servo.Jog2) THEN #Man."Step" := 0; END_IF;
   #_w2 := "AlwaysTRUE" AND (#Man."Step" = 10) AND #iMotionPermit;
   IF #_w2 THEN #Auto."Step" := 0; END_IF;
   #"Timer".T7.TON(IN := #_w2, PT := T#100ms);
   IF #"Timer".T7.Q THEN #Man."Step" := 20; END_IF;
   #Man.GoAbs := "AlwaysTRUE" AND (#Man."Step" = 20);
   IF #Man.GoAbs AND #Servo.SoftPosOK THEN #Man."Step" := 0; END_IF;
END_REGION

REGION Network 8: Premission Alarm
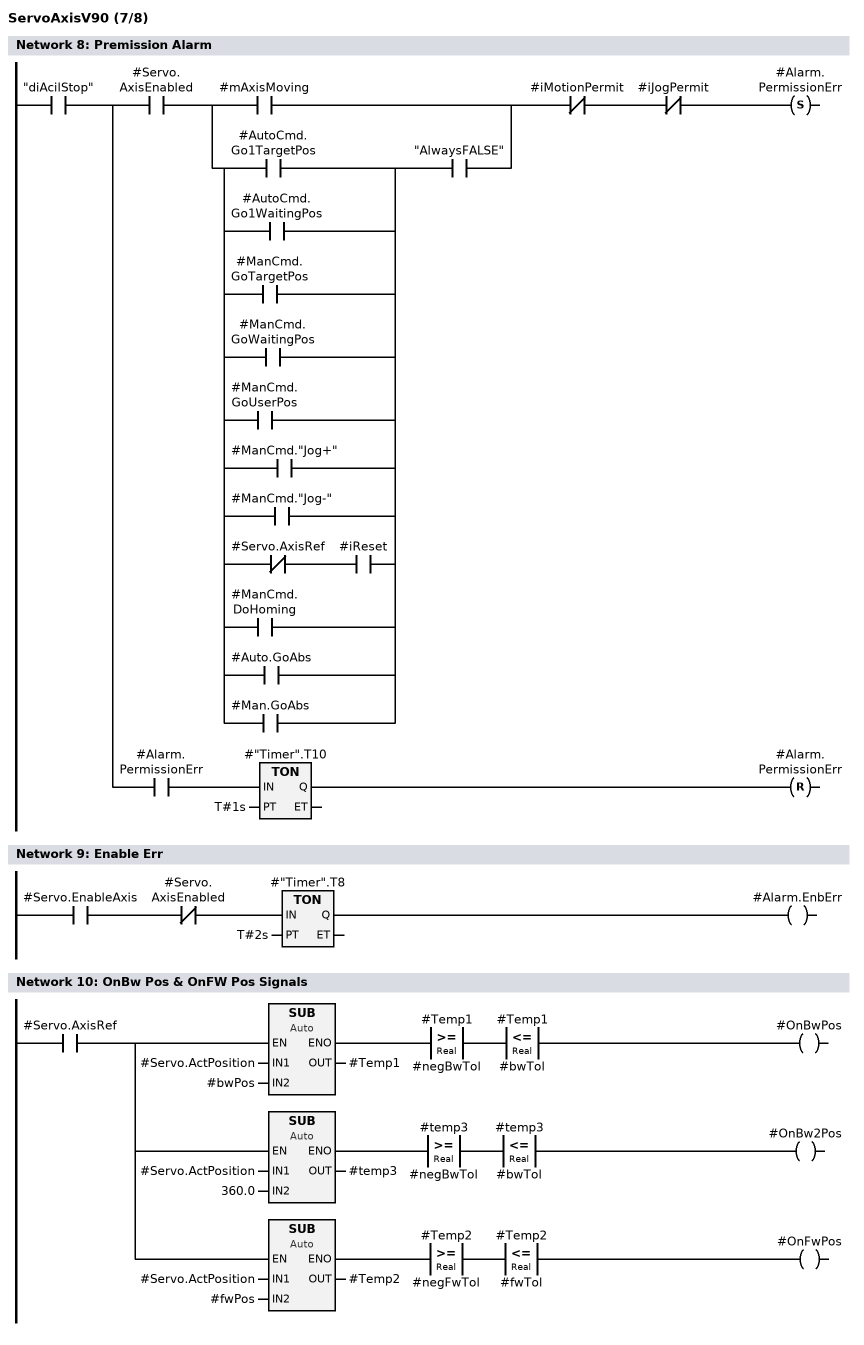
   IF "diAcilStop" AND #Servo.AxisEnabled AND (#mAxisMoving OR ((#AutoCmd.Go1TargetPos OR #AutoCmd.Go1WaitingPos OR #ManCmd.GoTargetPos OR #ManCmd.GoWaitingPos OR #ManCmd.GoUserPos OR #ManCmd."Jog+" OR #ManCmd."Jog-" OR (NOT #Servo.AxisRef AND #iReset) OR #ManCmd.DoHoming OR #Auto.GoAbs OR #Man.GoAbs) AND "AlwaysFALSE")) AND NOT #iMotionPermit AND NOT #iJogPermit THEN
       #Alarm.PermissionErr := TRUE;
   END_IF;
   #"Timer".T10.TON(IN := "diAcilStop" AND #Alarm.PermissionErr, PT := T#1s);
   IF #"Timer".T10.Q THEN #Alarm.PermissionErr := FALSE; END_IF;
END_REGION

REGION Network 9: Enable Err
   #"Timer".T8.TON(IN := #Servo.EnableAxis AND NOT #Servo.AxisEnabled, PT := T#2s);
   #Alarm.EnbErr := #"Timer".T8.Q;
END_REGION

REGION Network 10: OnBw Pos & OnFW Pos Signals
   RUNG wire#powerrail
      Contact( #Servo.AxisRef )
      wire#w1
      Sub(in1 := #Servo.ActPosition, in2 := #bwPos, out => #Temp1)
      { S7_Templates := "SrcType := Real" } GE_Contact(in1 := #Temp1, in2 := #negBwTol)
      { S7_Templates := "SrcType := Real" } LE_Contact(in1 := #Temp1, in2 := #bwTol)
      Coil( #OnBwPos )
   END_RUNG
   RUNG wire#w1
      Sub(in1 := #Servo.ActPosition, in2 := 360.0, out => #temp3)
      { S7_Templates := "SrcType := Real" } GE_Contact(in1 := #temp3, in2 := #negBwTol)
      { S7_Templates := "SrcType := Real" } LE_Contact(in1 := #temp3, in2 := #bwTol)
      Coil( #OnBw2Pos )
   END_RUNG
   RUNG wire#w1
      Sub(in1 := #Servo.ActPosition, in2 := #fwPos, out => #Temp2)
      { S7_Templates := "SrcType := Real" } GE_Contact(in1 := #Temp2, in2 := #negFwTol)
      { S7_Templates := "SrcType := Real" } LE_Contact(in1 := #Temp2, in2 := #fwTol)
      Coil( #OnFwPos )
   END_RUNG
   // the same network as SCL:
   IF #Servo.AxisRef THEN #Temp1 := #Servo.ActPosition - #bwPos; END_IF;
   #OnBwPos := #Servo.AxisRef AND (#Temp1 >= #negBwTol) AND (#Temp1 <= #bwTol);
   IF #Servo.AxisRef THEN #temp3 := #Servo.ActPosition - 360.0; END_IF;
   #OnBw2Pos := #Servo.AxisRef AND (#temp3 >= #negBwTol) AND (#temp3 <= #bwTol);
   IF #Servo.AxisRef THEN #Temp2 := #Servo.ActPosition - #fwPos; END_IF;
   #OnFwPos := #Servo.AxisRef AND (#Temp2 >= #negFwTol) AND (#Temp2 <= #fwTol);
END_REGION

REGION Network 11
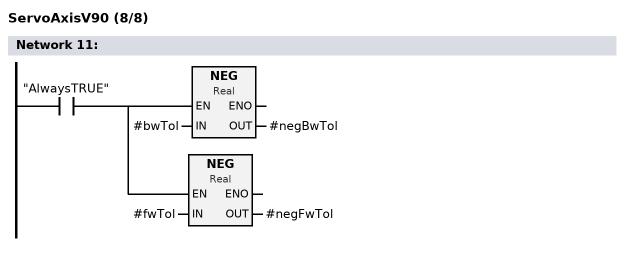
   RUNG wire#powerrail
      Contact( "AlwaysTRUE" )
      wire#w1
      { S7_Templates := "SrcType := Real" } Neg(in := #bwTol, out => #negBwTol)
   END_RUNG
   RUNG wire#w1
      { S7_Templates := "SrcType := Real" } Neg(in := #fwTol, out => #negFwTol)
   END_RUNG
   // the same network as SCL:
   IF "AlwaysTRUE" THEN
       #negBwTol := -#bwTol;
       #negFwTol := -#fwTol;
   END_IF;
END_REGION
END_FUNCTION_BLOCK

// ===== library: MasterCopy "ManServo" =====

TYPE "ManServo"
   STRUCT
      GoTargetPos : Bool;
      GoWaitingPos : Bool;
      GoUserPos : Bool;
      DoHoming : Bool;
      "Jog+" : Bool;
      "Jog-" : Bool;
      UserPos : Real;
      UserSpeed : Int;
   END_STRUCT;
END_TYPE

// ===== library: MasterCopy "fbValf" =====

// folder: Valf

FUNCTION_BLOCK "fbValf"   // FB1000, SCL
TITLE = Pnömatik Valf
{ S7_Optimized_Access := 'FALSE' }
AUTHOR : OrhunÇ
FAMILY : 1200
NAME : 1
VERSION : 0.1
// Pnömatik valf  ve iş elemanları için yazılmıştır
   VAR_INPUT
      iTip : Int := 1;   // 1: Çift Etkili Çift Sensör, 2:Tek Etkili Çift Sensör 3:Çift Etkili Sensörsüz 4:Tek Etkili Sensörsüz 5:Çift Etkili 3 Konumlu Sensörlü
      iGüvenlik : Bool := true;   // Güvenlik biti; Acil stop, ışık bariyeri ve piston güvenli hareket bilgileri vb.
      iMan : Bool := false;   // Manuel :Bit Setlendiğinde piston manuelde çalıştırılır.
      iManIleri : Bool := false;   // Manuelde Ileri Komutu
      iManGeri : Bool := false;   // Manulede geri Komutu
      iOto : Bool := false;   // Otomatik:Bit Setlendiğinde piston otomatikte çalıştırılır.
      iOtoIleri : Bool := false;   // Otomatikte ileri Komutu
      iOtoGeri : Bool := false;   // Otomatikte Geri Komutu
      iIleriSens : Bool := false;   // Otomatik Ileri Komutu Tip 3 ve4'te Kullanılmaz
      iGeriSens : Bool := false;   // Otomatik Geri Komutu Tip 3 ve 4'e Kullanılmaz
      iReset : Bool := false;   // Hata Reset
      iParam : Struct   // Fonksiyon Parametreleri
         hataZmni : Time := T#10S;   // Belirtilen zaman aralığında piston hareketini tamamlamaz ise(Geri veya Ileri) ilgili hata setlenir.Tip3 ve 4'te Kullanılmaz
         ileriBaskiZmni : Time := T#1s;   // 5/3 Pnömatik veya Hidrolik Valflerde ileri baskı süresi
         geriBaskiZmni : Time := T#1s;   // 5/3 Pnömatik veya Hidrolik Valflerde Geri baskı süresi
         manMod : Bool := false;   // Manuel Mod(5/3 Pnömatik veya Hidrolik Valfler için) false: buton basılı iken işlem görür, true: buton trig ile hareket tamamlanır.
      END_STRUCT;
   END_VAR
   VAR_OUTPUT
      oIleri : Bool := false;   // Piston Ileri Komutu
      oGeri : Bool := false;   // Piston Geri Komutu. Tip 2 ve 4 te kullanılmaz.
      oIleriHrktOk : Bool := false;   // Piston Ileri Hareketi sorunsuz tamamlandığında bit setlenir.Tip 3 ve 4'te Kullanılmaz
      oGeriHrktOk : Bool := false;   // Piston Geri Hareketi sorunsuz tamamlandığında bit setlenir.Tip 3 ve 4'te Kullanılmaz
      oHata : Array[0..4] of Bool;   // 0-Ileri Hata;1-GeriHata;2-Both Sensors Are Not Activated Uyarısı;3-Safety Fault;4-iki sensör görüyor / 0-Ileri Hata;1-GeriHata;2-Sensörler Görmüyor Uyarısı;3-Güvenlik Ihlali;4-iki sensör görüyor
   END_VAR
   VAR
      sManHareketIleri : Bool := false;   // Manuel Ileri Hareket
      sManHareketGeri : Bool := false;   // Manuel Geri Hareket
      sOtoHareketGeri : Bool := false;   // Otomatik Ileri Hareket
      sOtoHareketIleri : Bool := false;   // Otomatik Geri Hareket
      sGeriHata : Bool := false;   // Geri hatası için ayrıca kullanılan değişken
      sIleriHata : Bool := false;   // Ileri hatası için ayrıca kullanılan değişken
      sTGeriHarHata : TON_TIME;   // Geri Hareket Hata Bekleme
      sTIleriHarHata : TON_TIME;   // Ileri Hareket Hata Bekleme
      sTGeriSens : TON_TIME;   // Geri Sensör Hatası
      sTIleriSens : TON_TIME;   // Ileri Sensör Hatası
      sTSensHata : TON_TIME;   // Herhangi bir sensör görmediğinde oluşacak hata(sensörlü tiplerde)
      sTOFIleri : TOF_TIME;   // Tip 5 'te ileri hareketin tamamlanmasından sonraki baskı süresi
      sTOFIleri_q : Bool;   // Tof Çıkış
      sTOFGeri : TOF_TIME;   // Tip 5 'te Geri hareketin tamamlanmasından sonraki baskı süresi
      sTOFGeri_q : Bool := false;   // Tof Çıkış
      sHataVar : Bool := false;   // Hata Varlık bilgisi
      IEC_Timer_0_Instance : TON_TIME;   // İki sensörde aynı anda gördüğünde hata için bekleme süresi
      IEC_Timer_1_Instance : TON_TIME;
      IEC_Timer_0_Instance_q : Bool;   // İki sensör hata süresi çıkışı
      IEC_Timer_1_Instance_1 : Bool;
   END_VAR
   VAR_TEMP
      i : Int;   // değişken
   END_VAR
BEGIN
   (* Hata Açıklamaları
   oHata[0]; İleri hareket hatası
   oHata[1]; Geri hareket hatası
   oHata[2]; Sensörler görmüyor uyarısı
   oHata[3]; Güvenlik İhlali
   oHata[4]; İki Sensörde Görüyor Hatası
   *)

   //Tip Seçimi
   CASE #iTip OF
       1:
           GOTO Tip1;//Çift Bobinli Çift Sensörlü tip
       2:
           GOTO Tip2;//Tek Bobinli(Yay Geri Dönüşlü)Çift Sensörlü tip 
       3:
           GOTO Tip3;//Çift Bobinli (5/3 Valf ve hidrolik) Sensörsüz Tip
       4:
           GOTO Tip4;//Tek Bobinli Sensörsüz Tip
       5:
           GOTO Tip5;//Çift Bobinli (5/3 Valf ve hidrolik) Çift Sensörlü
   END_CASE;

   //---------------------------------------------------------------------------------------------------------------------------------------------------------------------
   /////////////////////////////////////ÇİFT BOBİNLİ ÇİFT SENSÖRLÜ PİSTON//////////////////

   Tip1:;
   //Manuel Hareket Komutları 
   IF #iGüvenlik AND #iMan THEN
       //Geri
       IF #iManGeri THEN
           #sManHareketGeri := TRUE;
           #sManHareketIleri := FALSE;
       END_IF;
       //İleri
       IF #iManIleri THEN
           #sManHareketIleri := TRUE;
           #sManHareketGeri := FALSE;
       END_IF;
   ELSE
       #sManHareketGeri := FALSE;
       #sManHareketIleri := FALSE;
   END_IF;


   //Otomatik Hareket Komutları
   IF #iGüvenlik AND #iOto THEN
       //Geri
       IF #iOtoGeri THEN
           #sOtoHareketGeri := TRUE;
           #sOtoHareketIleri := FALSE;
       END_IF;
       //İleri
       IF #iOtoIleri THEN
           #sOtoHareketIleri := TRUE;
           #sOtoHareketGeri := FALSE;
       END_IF;
   ELSE
       #sOtoHareketGeri := FALSE;
       #sOtoHareketIleri := FALSE;
   END_IF;

   //Otomatik Ve manuel hareketlerin fiziksel çıkışlara aktarılması.
   #oGeri := (#sManHareketGeri OR #sOtoHareketGeri) AND NOT (#iGeriSens AND NOT #sGeriHata) AND NOT #sHataVar;

   //Geri Sensörünün algılanması
   #sTGeriSens(IN := #iGeriSens,
               PT := t#5750ms);
   IF #sTGeriSens.Q THEN
       #sManHareketGeri := FALSE;
       #sOtoHareketGeri := FALSE;
   END_IF;

   #oIleri := (#sManHareketIleri OR #sOtoHareketIleri) AND NOT (#iIleriSens AND NOT #sIleriHata) AND NOT #sHataVar;

   //İleri Sensörünün algılanması
   #sTIleriSens(IN := #iIleriSens,
                PT := t#5750ms);
   IF #sTIleriSens.Q THEN
       #sManHareketIleri := FALSE;
       #sOtoHareketIleri := FALSE;
   END_IF;

   //Hareket Tamamlandı bilgileri
   #oGeriHrktOk := #iGeriSens AND NOT #sGeriHata;
   #oIleriHrktOk := #iIleriSens AND NOT #sIleriHata;

   //Alarmlar
   //Geri hareket hatası
   #sTGeriHarHata(IN := NOT #iReset AND (#sManHareketGeri OR #sOtoHareketGeri) AND NOT #iGeriSens,
                  PT := #iParam.hataZmni,
                  Q => #sGeriHata);
   #oHata[1] := #sGeriHata;

   //İleri hareket hatası
   #sTIleriHarHata(IN := NOT #iReset AND (#sManHareketIleri OR #sOtoHareketIleri) AND NOT #iIleriSens,
                   PT := #iParam.hataZmni,
                   Q => #sIleriHata);
   #oHata[0] := #sIleriHata;

   //Belirli süre sonunda sensörlerin görmemesi uyarısı-Sensörlü tiplerde
   #sTSensHata(IN := NOT #oGeriHrktOk AND NOT #oIleriHrktOk AND NOT #iReset,
               PT := #iParam.hataZmni * 2);//Hata zamanın 3 katı)
   IF #sTSensHata.Q THEN
       #oHata[2] := TRUE;
   END_IF;

   //İki sensöründe aynı anda görmesi hatası(Sensörlerin bozulması durumunda meydana çıkar)
   #IEC_Timer_1_Instance(IN := #iGeriSens AND #iIleriSens,
                         PT := t#1s,
                         Q => #IEC_Timer_1_Instance_1);


   IF #IEC_Timer_1_Instance_1 THEN 
       #oHata[4] := TRUE;
   END_IF;

   GOTO SON;
   //---------------------------------------------------------------------------------------------------------------------------------------------------------------------
   /////////////////////////////////////TEK BOBİNLİ ÇİFT SENSÖRLÜ PİSTON///////////////////
   Tip2:;
   //Manuel Hareket Komutları 
   IF #iGüvenlik AND #iMan THEN
       //Geri
       IF #iManGeri THEN
           #sManHareketIleri := FALSE;
       END_IF;
       //İleri
       IF #iManIleri THEN
           #sManHareketIleri := TRUE;
       END_IF;
   ELSE
       #sManHareketIleri := FALSE;
       #sManHareketGeri := FALSE;
   END_IF;

   //Otomatik Hareket Komutları
   IF #iGüvenlik AND #iOto THEN
       //Geri 
       IF #iOtoGeri THEN
           #sOtoHareketIleri := FALSE;
       END_IF;
       //İleri
       IF #iOtoIleri THEN
           #sOtoHareketIleri := TRUE;
       END_IF;
   ELSE
       #sOtoHareketIleri := FALSE;
       #sOtoHareketGeri := FALSE;
   END_IF;

   //Otomatik Ve manuel hareketlerin fiziksel çıkışlara aktarılması.
   #oIleri := (#sManHareketIleri OR #sOtoHareketIleri);

   //Hareket Tamamlandı bilgileri
   #oGeriHrktOk := #iGeriSens AND NOT #sGeriHata;
   #oIleriHrktOk := #iIleriSens AND NOT #sIleriHata;

   //Alarmlar
   //Geri hareket hatası
   #sTGeriHarHata(IN := NOT #iReset AND NOT (#sManHareketIleri OR #sOtoHareketIleri) AND NOT #iGeriSens,
                  PT := #iParam.hataZmni,
                  Q => #sGeriHata);
   #oHata[1] := #sGeriHata;

   //İleri Hareket Hatası
   #sTIleriHarHata(IN := NOT #iReset AND (#sManHareketIleri OR #sOtoHareketIleri) AND NOT #iIleriSens,
                   PT := #iParam.hataZmni,
                   Q => #sIleriHata);
   #oHata[0] := #sIleriHata;

   //Belirli süre sonunda sensörlerin görmemesi uyarısı-Sensörlü tiplerde
   #sTSensHata(IN := NOT #iReset AND NOT #oGeriHrktOk AND NOT #oIleriHrktOk,
               PT := #iParam.hataZmni * 3);//Hata zamanın 3 katı)
   IF #sTSensHata.Q THEN
       #oHata[2] := TRUE;
   END_IF;

   //İki sensöründe aynı anda görmesi hatası(Sensörlerin bozulması durumunda meydana çıkar)
   IF #iGeriSens AND #iIleriSens THEN
       #oHata[4] := TRUE;
   END_IF;

   GOTO SON;
   //---------------------------------------------------------------------------------------------------------------------------------------------------------------------
   /////////////////////////////////////ÇİFT BOBİNLİ 5/3 PNOMATİK İLE HİDROLİK VALF VE SENSÖRSÜZ PİSTON//////////////////////
   Tip3:;
   //Manuel Hareket Komutları
   IF #iGüvenlik AND #iMan THEN
       //Geri
       #sManHareketGeri := #iManGeri;
       //İleri
       #sManHareketIleri := #iManIleri;
       //Otomatik Statiklerin resetlenmesi
       #sOtoHareketGeri := FALSE;
       #sOtoHareketIleri := FALSE;
   END_IF;

   //Otomatik Hareket Komutları
   IF #iGüvenlik AND #iOto THEN
       //Geri 
       #sOtoHareketGeri := #iOtoGeri;
       //İleri
       #sOtoHareketIleri := #iOtoIleri;
       //Manuel Statiklerin resetlenmesi
       #sManHareketGeri := FALSE;
       #sManHareketIleri := FALSE;
   END_IF;
   //Otomatik Ve manuel hareketlerin fiziksel çıkışlara aktarılması.
   #oGeri := #sManHareketGeri OR #sOtoHareketGeri;
   #oIleri := #sManHareketIleri OR #sOtoHareketIleri;

   //Alarmlar

   //Kullanılmayan çıkış bitlerinin resetlenmesi
   #oGeriHrktOk := FALSE;
   #oIleriHrktOk := FALSE;
   #oHata[0] := FALSE;
   #oHata[1] := FALSE;
   #oHata[2] := FALSE;
   #oHata[4] := FALSE;

   GOTO SON;
   //---------------------------------------------------------------------------------------------------------------------------------------------------------------------
   /////////////////////////////////////TEK BOBİNLİ SENSÖRSÜZ PİSTON///////////////////
   Tip4:;
   //Manuel Hareket Komutları 
   IF #iGüvenlik AND #iMan THEN
       //Geri
       IF #iManGeri AND NOT #iManIleri THEN
           #sManHareketIleri := FALSE;
       END_IF;
       //İleri
       IF #iManIleri AND NOT #iManGeri THEN
           #sManHareketIleri := TRUE;
       END_IF;
       #sOtoHareketIleri := FALSE;
       #sOtoHareketGeri := FALSE;
   END_IF;

   //Otomatik Hareket Komutları
   IF #iGüvenlik AND #iOto THEN
       //Geri 
       IF #iOtoGeri AND NOT #iOtoIleri THEN
           #sOtoHareketIleri := FALSE;
       END_IF;
       //İleri
       IF #iOtoIleri AND NOT #iOtoGeri THEN
           #sOtoHareketIleri := TRUE;
       END_IF;
       #sManHareketIleri := FALSE;
       #sManHareketGeri := FALSE;
   END_IF;
   //Otomatik Ve manuel hareketlerin fiziksel çıkışlara aktarılması.
   #oIleri := #sManHareketIleri OR #sOtoHareketIleri;


   //Kullanılmayan çıkış bitlerinin resetlenmesi
   #oGeriHrktOk := FALSE;
   #oIleriHrktOk := FALSE;
   #oHata[0] := FALSE;
   #oHata[1] := FALSE;
   #oHata[2] := FALSE;
   #oHata[4] := FALSE;

   GOTO SON;

   //---------------------------------------------------------------------------------------------------------------------------------------------------------------------
   ///////////////ÇİFT BOBİNLİ KAPALI VEYA AÇIK MERKEZ VALF ÇİFT SENSÖRLÜ PİSTON////////////////
   Tip5:;
   //Manuel Hareket Komutları
   //Mode:SetBit
   IF #iParam.manMod THEN
       IF #iGüvenlik AND #iMan THEN
           //Geri
           IF #iManGeri THEN
               #sManHareketGeri := TRUE;
               #sManHareketIleri := FALSE;
           END_IF;
           //İleri
           IF #iManIleri THEN
               #sManHareketIleri := TRUE;
               #sManHareketGeri := FALSE;
           END_IF;
       ELSE
           #sManHareketGeri := FALSE;
           #sManHareketIleri := FALSE;
       END_IF;
   ELSE
       //Mode:SetBitWhileKeyPressed
       IF #iGüvenlik AND #iMan THEN
           //Geri
           #sManHareketGeri := #iManGeri;
           //İleri
           #sManHareketIleri := #iManIleri;
           //Otomatik Statiklerin resetlenmesi
           #sOtoHareketGeri := FALSE;
           #sOtoHareketIleri := FALSE;
       END_IF;
   END_IF;

   //Otomatik Hareket Komutları
   IF #iGüvenlik AND #iOto THEN
       //Geri
       IF #iOtoGeri THEN
           #sOtoHareketGeri := TRUE;
           #sOtoHareketIleri := FALSE;
       END_IF;
       //İleri
       IF #iOtoIleri THEN
           #sOtoHareketIleri := TRUE;
           #sOtoHareketGeri := FALSE;
       END_IF;
   ELSE
       #sOtoHareketGeri := FALSE;
       #sOtoHareketIleri := FALSE;
   END_IF;




   //Otomatik Ve manuel hareketlerin fiziksel çıkışlara aktarılması.
   //Geri Sensörü gördükten 1 saniye sonra baskı bırakılır.
   #sTOFGeri(IN := ((#sManHareketGeri AND #iParam.manMod) OR #sOtoHareketGeri) AND NOT (#iGeriSens AND NOT #sGeriHata) AND NOT #sHataVar,
             PT :=#iParam.geriBaskiZmni,
             Q => #sTOFGeri_q);
   //Belirli zaman sonunda Çıkış Kesilir
   #oGeri := #sTOFGeri_q OR (#sManHareketGeri AND NOT #iParam.manMod);

   //Geri Sensörünün algılanması
   #sTGeriSens(IN := #iGeriSens,
               PT := t#5750ms);
   IF #sTGeriSens.Q THEN
       #sManHareketGeri := FALSE;
       #sOtoHareketGeri := FALSE;
   END_IF;

   //İLERİ HAREKET
   //İleri Sensörü gördükten belirli saniye sonra baskı bırakılır.
   #sTOFIleri(IN := ((#sManHareketIleri AND #iParam.manMod)OR #sOtoHareketIleri) AND NOT (#iIleriSens AND NOT #sIleriHata) AND NOT #sHataVar,
              PT := #iParam.ileriBaskiZmni,
              Q => #sTOFIleri_q);

   //Belirli zaman sonunda Çıkış Kesilir
   #oIleri := #sTOFIleri_q OR (#sManHareketIleri AND NOT #iParam.manMod);

   //İleri Sensörünün algılanması
   #sTIleriSens(IN := #iIleriSens,
                PT := t#5750ms);
   IF #sTIleriSens.Q THEN
       #sManHareketIleri := FALSE;
       #sOtoHareketIleri := FALSE;
   END_IF;


   //Hareket Tamamlandı bilgileri
   #oGeriHrktOk := #iGeriSens AND NOT #sGeriHata AND NOT #oGeri;
   #oIleriHrktOk := #iIleriSens AND NOT #sIleriHata AND NOT #oIleri;

   //Alarmlar
   //Geri hareket hatası
   #sTGeriHarHata(IN := NOT #iReset AND (#sManHareketGeri OR #sOtoHareketGeri) AND NOT #iGeriSens,
                  PT := #iParam.hataZmni,
                  Q => #sGeriHata);
   #oHata[1] := #sGeriHata;

   //İleri hareket hatası
   #sTIleriHarHata(IN := NOT #iReset AND (#sManHareketIleri OR #sOtoHareketIleri) AND NOT #iIleriSens,
                   PT := #iParam.hataZmni,
                   Q => #sIleriHata);
   #oHata[0] := #sIleriHata;

   //Belirli süre sonunda sensörlerin görmemesi uyarısı-Sensörlü tiplerde
   #sTSensHata(IN := NOT #oGeriHrktOk AND NOT #oIleriHrktOk AND NOT #iReset,
               PT := #iParam.hataZmni * 2);//Hata zamanın 3 katı)
   IF #sTSensHata.Q THEN
       #oHata[2] := TRUE;
   END_IF;

   //İki sensöründe aynı anda görmesi hatası(Sensörlerin bozulması durumunda meydana çıkar)
   #IEC_Timer_0_Instance(IN:=#iGeriSens AND #iIleriSens,
                         PT:=t#1s,
                         Q=>#IEC_Timer_0_Instance_q);

   IF #IEC_Timer_0_Instance_q THEN
       #oHata[4] := TRUE;
   END_IF;

   SON:;
   //ORtak Alarmlar
   //güvenlik ihlal uyarısı
   IF NOT #iGüvenlik AND (#iMan AND (#iManIleri OR #iManGeri) OR (#iOto AND (#iOtoIleri OR #iOtoGeri))) THEN
       #oHata[3] := TRUE;
   END_IF;

   //Reset
   IF #iReset AND #sHataVar THEN
       #sManHareketGeri := FALSE;
       #sManHareketIleri := FALSE;
       #sOtoHareketGeri := FALSE;
       #sOtoHareketIleri := FALSE;
       FOR #i := 0 TO 4 DO
           #oHata[#i] := FALSE;
       END_FOR;
       #sHataVar := FALSE;
   END_IF;

   //Hata var biti

   FOR #i := 0 TO 4 DO
       IF #oHata[#i] = TRUE THEN
           #sHataVar := TRUE;
       END_IF;
   END_FOR;
END_FUNCTION_BLOCK

// ===== library: MasterCopy "udtValf" =====

TYPE "udtValf"
VERSION : 0.1
   STRUCT
      in : Struct
         tip : Int := 1;   // Valf Tipi
         guv : Bool := true;   // Güvenlik komutu
         mİleri : Bool := false;   // Piston manuel ileri komutu
         mGeri : Bool := false;   // Piston manuel geri komutu
         oİleri : Bool := false;   // Piston otomatik ileri komutu
         oGeri : Bool := false;   // Piston otomatik geri komutu
         param : Struct   // Fonksiyon Parametreleri
            hataZmni : Time := T#10s;   // Belirtilen zaman aralığında piston hareketini tamamlamaz ise(Geri veya Ileri) ilgili hata setlenir.Tip3 ve 4'te Kullanılmaz
            ileriBaskiZmni : Time := T#1s;   // 5/3 Pnömatik veya Hidrolik Valflerde ileri baskı süresi
            geriBaskiZmni : Time := T#1s;   // 5/3 Pnömatik veya Hidrolik Valflerde Geri baskı süresi
            manMod : Bool := false;   // Manuel Mod(5/3 Pnömatik veya Hidrolik Valfler için) false: buton basılı iken işlem görür, true: buton trig ile hareket tamamlanır.
         END_STRUCT;
      END_STRUCT;
      out : Struct
         hata : Array[0..4] of Bool;   // Hata Bilgileri
         ileriHrktOk : Bool;   // İleri hareket tamamlandı
         geriHrktOk : Bool;   // Geri hareket tamamlandı
      END_STRUCT;
   END_STRUCT;
END_TYPE

// ===== library: MasterCopy "udtGraf" =====

TYPE "udtGraf"
VERSION : 0.1
   STRUCT
      idleC : Bool;   // Sistem boşta koşulları
      startC : Bool;   // Start koşulları
      startCmd : Bool;   // Start Komutu
      runStep : Bool;   // Adım çalıştırma
      st : Array[0..63] of Bool;   // Set Reset mantığı Adım
      tt : Array[0..63] of Bool;   // Set Reset mantığı Adım Aynalama
      "step" : Int;   // intiger Mantığı Ana Adım
      subStep : Array[1..10] of Int;   // İntiger Mantığı Alt Adımlar
   END_STRUCT;
END_TYPE